{attribute 'qualified_only'}
{attribute 'strict'}
TYPE E_CraneCommunicationType :
(
	EAP,
	TCP_IP
);
END_TYPE

(* stored: Version 1.1.0.1, ProductVersion 3.1.4024.9
   DUT E_CraneCommunicationType: Id {8816e2bb-8d6b-445d-b262-43292b3cec2f} *)
